TYPE OpticalPowermeterConfigs :
STRUCT
	PM101OpticalPowermeterConfigHs : PM101OpticalPowermeterConfig;
	PM101OpticalPowermeterConfigHt : PM101OpticalPowermeterConfig;
END_STRUCT
END_TYPE

(* stored: Version 1.1.0.1, ProductVersion 3.1.4024.3
   DUT OpticalPowermeterConfigs: Id {3814a299-5a5b-4e9f-9972-479d23426e6a} *)
